// Mitsubishi GX Works2 project: 14.05.24-cascade-2   PLC: FX3G
// Каскад начинается с 2х.

TYPE PUMP : STRUCT
  TurnOn : INT;
  EnableManual : INT;
  OutTask : INT;  (* AO value 0-4000 *)
  Blocked : INT;
  Enable : INT;
  ManualTask : INT;  (* Percent 0.0-100.0 *)
  EnableAuto : INT;
END_STRUCT END_TYPE

// global labels: GVL
VAR_GLOBAL
  giMaxTempr AT R0 : INT;
  gxManual AT M2000 : BOOL;
  gxAuto AT M400 : BOOL;
  gxReset AT M2002 : BOOL;
  gxPump1Enable AT M500 : BOOL;
  gxPump2Enable AT M501 : BOOL;
  gxPump3Enable AT M502 : BOOL;
  gxPump4Enable AT M503 : BOOL;
  gxPump5Enable AT M504 : BOOL;
  gxPump6Enable AT M505 : BOOL;
  arModbus : ARRAY [0..29] OF MB_REG;
  giPSV AT R1 : INT;  (* Set value for pressure 0.00 *)
  giPIDtask AT R2 : INT;
  gxPIDAT AT M2020 : BOOL;
  gxPIDATMode AT M2021 : BOOL;
  gxPump1Manual AT M2009 : BOOL;
  gxPump2Manual AT M2010 : BOOL;
  gxPump3Manual AT M2011 : BOOL;
  gxPump4Manual AT M2012 : BOOL;
  gxPump5Manual AT M2013 : BOOL;
  arPumps : ARRAY [0..4] OF PUMP;
END_VAR
VAR_GLOBAL CONSTANT
  c_PUMPS : INT := 5;
END_VAR
VAR_GLOBAL
  giMaxDiffPressure AT R3 : INT;
  gxPump6Manual AT M2014 : BOOL;
  giMinFlow AT R4 : INT;  (* Если проток больше чем это то включаем полив *)
  giMinPressure AT R5 : INT;  (* Если давление меньше чем это то включаем полив *)
  giMaxPressureRelease AT R6 : INT;
  gxValveManual AT M2015 : BOOL;
  gxErrorJokey AT M2016 : BOOL;
  gxIsAlarm AT M2017 : BOOL;
  gxRecord AT M2018 : BOOL;
  gxResetCounters AT M2019 : BOOL;
END_VAR

// global labels: IO
VAR_GLOBAL
  AI_T_Pump1 AT D0 : INT;
  AI_T_Pump2 AT D1 : INT;
  AI_T_Pump3 AT D2 : INT;
  AI_T_Pump4 AT D3 : INT;
  AI_T_Pump5 AT D4 : INT;
  AI_T_Pump6 AT D5 : INT;
  AI_P_Collector AT D6 : INT;
  AI_P_Filter AT D7 : INT;
  AI_F_Flow AT D8 : INT;
  DI_HighPressure AT X000 : BOOL;
  DI_AU AT X001 : BOOL;
  DI_RKF AT X002 : BOOL;
  DI_T_Panel1_High AT X003 : BOOL;
  DI_T_Panel2_High AT X004 : BOOL;
  DI_FlowPLS AT X005 : BOOL;
  DI_FlowPump1 AT X012 : BOOL;
  DI_FlowPump2 AT X013 : BOOL;
  DI_FlowPump3 AT X014 : BOOL;
  DI_FlowPump4 AT X015 : BOOL;
  DI_FlowPump5 AT X016 : BOOL;
  DI_FlowPump6 AT X017 : BOOL;
  DO_Pump1 AT Y004 : BOOL;
  DO_ResetVFD1 AT Y005 : BOOL;
  DO_Pump2 AT Y006 : BOOL;
  DO_ResetVFD2 AT Y007 : BOOL;
  DO_Pump3 AT Y010 : BOOL;
  DO_ResetVFD3 AT Y011 : BOOL;
  DO_Pump4 AT Y012 : BOOL;
  DO_ResetVFD4 AT Y013 : BOOL;
  DO_Pump5 AT Y014 : BOOL;
  DO_ResetVFD5 AT Y015 : BOOL;
  DO_PumpJok AT Y016 : BOOL;
  DO_ResetVFDJok AT Y017 : BOOL;
  DO_ReleaseValve AT Y020 : BOOL;
  AO_Pump1 AT D8050 : INT;
  AO_Pump2 AT D8051 : INT;
  AO_Pump3 AT D8052 : INT;
  AO_Pump4 AT D8053 : INT;
  AO_Pump5 AT D8054 : INT;
END_VAR

// task INIT (event M8002, interval 0, priority 24): Init
// task PRC (event FALSE, interval T#50ms, priority 29): Process
// task Task_01 (event TRUE, interval 0, priority 31): POU_01
// user libraries (not included): AlarmManger128, Modbus, PumpControl, TimeControl, Utils

PROGRAM Init
VAR
  fbAmInit : AM_INIT;
END_VAR
(* Init PID *) (* Настройка параметров ПИД регулирования *)
R500 := 100; (* Time 1c *)
R501 := 2#0000_0000_0000_0001; (* Heating mode *)
R522 := 1000; (* Output max 100% *)
R523 := 0; (* Output min *)
R525 := 10; (* Delta for Autotune 0.5 bar *)
R526 := R522; (* Autotune output upper value *)
R527 := 0; (* Autotune output lower value *)

(* Start alarm manager data at D3000 *)
AM_D_START := 3000;

(* Temperature sensor 1-6 wire out *)
fbAmInit(iNum := 0, iSeverity := AM_ERROR, iProcess := 1);
fbAmInit(iNum := 1);
fbAmInit(iNum := 2);
fbAmInit(iNum := 3);
fbAmInit(iNum := 4);
fbAmInit(iNum := 5);
(* Pressure sensor wire out *)
fbAmInit(iNum := 6, xLock := 1);
(* Pressure sensor after filter wire out *)
fbAmInit(iNum := 7);
(* Flow meter wire out *)
fbAmInit(iNum := 8);
(* Alarm water level level *)
fbAmInit(iNum := 9);
(* Pump temperature too high *)
fbAmInit(iNum := 10, xLatch := 1, xLock := 0);
fbAmInit(iNum := 11);
fbAmInit(iNum := 12);
fbAmInit(iNum := 13);
fbAmInit(iNum := 14);
fbAmInit(iNum := 15);
(* Pump flow *)
fbAmInit(iNum := 16);
fbAmInit(iNum := 17);
fbAmInit(iNum := 18);
fbAmInit(iNum := 19);
fbAmInit(iNum := 20);
fbAmInit(iNum := 21);

(* Max pressure diff *)
fbAmInit(iNum := 22, xLatch := 1, xLock := 1);
(* High pressure *)
fbAmInit(iNum := 23, xLatch := 0, xLock := 1);
(* High tempr 1 *)
fbAmInit(iNum := 24, xLatch := 1, xLock := 1);
(* High tempr 2 *)
fbAmInit(iNum := 25, xLatch := 1, xLock := 1);
(* RKF *)
fbAmInit(iNum := 26, xLatch := 0, xLock := 1);
(* MB Timeout *)
fbAmInit(iNum := 27, xLatch := 0, xLock := 0);
(* Parametrs all set *)
fbAmInit(iNum := 28, xLatch := 0, xLock := 1);

(* Pump VFD Alarm *)
fbAmInit(iNum := 29, xLatch := 0, xLock := 0);
fbAmInit(iNum := 30);
fbAmInit(iNum := 31);
fbAmInit(iNum := 32);
fbAmInit(iNum := 33);
fbAmInit(iNum := 34);

(* Библиотека драйверов Modbus RTU , ПЛК Coolmay FX3G для управления преобразователями частоты , далее ПЧ *)
arModbus[0].iDev := H1; (* Device address *)
arModbus[0].iRDevNum := 3000; (* R memmory to locate result *)
arModbus[0].iNum := 14; (* Number of registers *)
arModbus[0].iReg := H3000; (* Modbus register *)
arModbus[0].iRF := H3; (* Read function *)
arModbus[0].iWR := MB_READ; (* Read and\or write access *)
arModbus[0].tCycle := T#1000ms; (* How oftent *)

arModbus[1].iDev := H2; (* Device address *)
arModbus[1].iRDevNum := 3020; (* R memmory to locate result *)
arModbus[1].iNum := 14; (* Number of registers *)
arModbus[1].iReg := H3000; (* Modbus register *)
arModbus[1].iRF := H3; (* Read function *)
arModbus[1].iWR := MB_READ; (* Read and\or write access *)
arModbus[1].tCycle := T#1000ms; (* How oftent *)

arModbus[2].iDev := H3; (* Device address *)
arModbus[2].iRDevNum := 3040; (* R memmory to locate result *)
arModbus[2].iNum := 14; (* Number of registers *)
arModbus[2].iReg := H3000; (* Modbus register *)
arModbus[2].iRF := H3; (* Read function *)
arModbus[2].iWR := MB_READ; (* Read and\or write access *)
arModbus[2].tCycle := T#1000ms; (* How oftent *)

arModbus[3].iDev := H4; (* Device address *)
arModbus[3].iRDevNum := 3060; (* R memmory to locate result *)
arModbus[3].iNum := 14; (* Number of registers *)
arModbus[3].iReg := H3000; (* Modbus register *)
arModbus[3].iRF := H3; (* Read function *)
arModbus[3].iWR := MB_READ; (* Read and\or write access *)
arModbus[3].tCycle := T#1000ms; (* How oftent *)

arModbus[4].iDev := H5; (* Device address *)
arModbus[4].iRDevNum := 3080; (* R memmory to locate result *)
arModbus[4].iNum := 14; (* Number of registers *)
arModbus[4].iReg := H3000; (* Modbus register *)
arModbus[4].iRF := H3; (* Read function *)
arModbus[4].iWR := MB_READ; (* Read and\or write access *)
arModbus[4].tCycle := T#1000ms; (* How oftent *)

arModbus[5].iDev := H6; (* Device address *)
arModbus[5].iRDevNum := 3100; (* R memmory to locate result *)
arModbus[5].iNum := 1; (* Number of registers *)
arModbus[5].iReg := H3002; (* Modbus register *)
arModbus[5].iRF := H4; (* Read function *)
arModbus[5].iWR := MB_READ; (* Read and\or write access *)
arModbus[5].tCycle := T#1000ms; (* How oftent *)
END_PROGRAM

PROGRAM POU_01
VAR
  iCount : INT;
  iCountEnabled : INT;
  iCountEbabledAuto : INT;
  iStep : INT;
  xAddOne : BOOL;
  xSubOne : BOOL;
  fbAmBlock : AM_IS_BLOCK;
  xError : BOOL;
  fbAmOrIsOn : AM_ORISON;
  fbReleaseTOF : TOF;
  fbRelease2TOF : TOF;
  iShifter : INT;
  iShifted : INT;
  xAfterAdd : BOOL;
  xFromJokey : BOOL;
  xAfterSub : BOOL;
END_VAR
IF MEP(gxAuto) AND gxPIDAT THEN
	R501 := 2#0000_0000_0011_0001; (* Autotune Step Response *)
	IF NOT gxPIDATMode THEN
		R501 := 2#0000_0000_0111_0001; (* Autotune limit cycle *)
	END_IF;
	gxPIDAT := FALSE;
END_IF;

RST(MEP(gxManual), gxAuto);
RST(MEP(gxAuto), gxManual);

fbAmBlock(iProcessNum := 1, iSeverity := AM_ERROR);
gxIsAlarm := fbAmBlock.Q;

(* IF there is blocking alarm AND we are in auto OR manual OR jokey mode, EXIT it *)
IF fbAmBlock.Q AND iStep <> 10 THEN	iStep := 0; END_IF;

PID(iStep = 30 AND (AI_P_Collector < (giPSV + 50)), giPSV, AI_P_Collector, R500, giPIDTask);

IF MEP(iStep = 30) THEN iShifter := INC5(iShifter); END_IF;
OUT_T(iStep = 30 AND xAfterAdd, TC14, 100);
RST(MEP(TS14), xAfterAdd);

OUT_T(iStep = 30 AND xAfterSub, TC16, 100);
RST(MEP(TS16), xAfterSub);

(*OUT_T(iStep = 30 AND NOT TS15 AND NOT xAfterAdd, TC15, 100);*)

OUT_T(iStep = 35, TC13, 60); (* time to add new pump *)
OUT_T(iStep = 30 AND AI_F_Flow < 200 AND (AI_P_Collector > giMinPressure), TC21, 50); (* to jokey *)

CASE iStep OF
	0: (* Init *)
		gxManual := FALSE;
		FOR iCount := 0 TO 4 DO
			arPumps[iCount].OutTask := 0;
			arPumps[iCount].TurnOn := 0;
			arPumps[iCount].ManualTask := 0;
			arPumps[iCount].EnableAuto := 0;
			arPumps[iCount].EnableManual := 0;
		END_FOR;
		iStep := 10;

	10: (* Idle *) (* *)
		IF gxManual AND NOT fbAmBlock.Q THEN
			iStep := 20;
		END_IF;
		IF gxAuto AND NOT fbAmBlock.Q THEN
			iStep := 30;
		END_IF;

	20: (* Manual *)
        FOR iCount := 0 TO 4 DO
			IF arPumps[iCount].Enable = 0 THEN arPumps[iCount].EnableManual := 0; END_IF;

			arPumps[iCount].TurnOn := BOOL_TO_INT(
				NOT INT_TO_BOOL(arPumps[iCount].Blocked)
				AND INT_TO_BOOL(arPumps[iCount].Enable)
				AND INT_TO_BOOL(arPumps[iCount].EnableManual)
			);

			arPumps[iCount].OutTask := 0;
			IF arPumps[iCount].TurnOn = 1 THEN
				arPumps[iCount].OutTask := SCALE(arPumps[iCount].ManualTask, 0, 1000, 0, 4000);
			END_IF;
		END_FOR;

		IF NOT gxManual THEN iStep := 0; END_IF;

	30: (* Auto CASCADE *)
		(* Once every 10 seconds *)
		iCountEnabled := 0;	 iCountEbabledAuto := 0;
		FOR iCount := 0 TO 4 DO
			IF arPumps[iCount].Enable = 0 THEN arPumps[iCount].EnableAuto := 0; END_IF;
			(* Globally ready pumps for work *)
			IF arPumps[iCount].Enable > 0 AND (arPumps[iCount].Blocked = 0) THEN
				iCountEnabled := iCountEnabled + 1;
			END_IF;

			(* Count currently enabled pumps in cascade *)
			iCountEbabledAuto := iCountEbabledAuto + arPumps[iCount].EnableAuto;
		END_FOR;
		
		(* Add new pump to cascade if PID task > 90.0% and there is a pump available *)
		xAddOne := xFromJokey OR ((giPIDTask > 950) AND (
			(iCountEbabledAuto > 0 AND AI_P_Collector < (giPSV - 100)) OR iCountEbabledAuto = 0
		) AND (iCountEnabled > iCountEbabledAuto));
		(* Subtract pump if task is less than 40.0% or 25 HGz if there are more than 2 pumps enabled *)
		xSubOne := giPIDTask < 780 AND iCountEbabledAuto > 2;
		xFromJokey := FALSE;
		
		IF xAddOne AND NOT xAfterAdd THEN 
			iStep := 35; 
		END_IF;
		
		FOR iCount := 0 TO 4 DO
			iShifted := SHFT(iShifter, iCount);
			IF xSubOne 
				AND NOT xAfterSub 
				AND arPumps[iShifted].Enable > 0 
				AND arPumps[iShifted].Blocked = 0 
				AND arPumps[iShifted].EnableAuto > 0 
			THEN
				arPumps[iShifted].EnableAuto := 0;
				xSubOne := FALSE;
				xAfterSub := TRUE;
			END_IF; 
			
			arPumps[iShifted].TurnOn := BOOL_TO_INT(
				NOT INT_TO_BOOL(arPumps[iShifted].Blocked) 
				AND INT_TO_BOOL(arPumps[iShifted].Enable) 
				AND INT_TO_BOOL(arPumps[iShifted].EnableAuto)
				AND AI_P_Collector < (giPSV + 50)
			);

			arPumps[iShifted].OutTask := 0;
			IF arPumps[iShifted].TurnOn > 0 THEN
				arPumps[iShifted].OutTask := SCALE(giPIDTask, 0, 1000, 0, 4000);
			END_IF;
		END_FOR;
		
		(* TODO condition to switch to Jokey *)
		
		(* IF AI_F_Flow <= giMinFlow THEN *) 
		IF  TS21 THEN 
			FOR iCount := 0 TO 4 DO
				arPumps[iCount].OutTask := 0;
				arPumps[iCount].TurnOn := 0;
				arPumps[iCount].ManualTask := 0;
				arPumps[iCount].EnableAuto := 0;
				arPumps[iCount].EnableManual := 0;
			END_FOR;
			iStep := 40;
		END_IF;

		IF NOT gxAuto OR gxReset THEN iStep := 0; END_IF;
	
	35:
	    iCountEbabledAuto := 0;
	    FOR iCount := 0 TO 4 DO
				iCountEbabledAuto := iCountEbabledAuto + arPumps[iCount].EnableAuto;
	    END_FOR;
	    
		FOR iCount := 0 TO 4 DO
			iShifted := SHFT(iShifter, iCount);
			IF xAddOne AND arPumps[iShifted].Enable > 0 AND arPumps[iShifted].Blocked = 0 AND arPumps[iShifted].EnableAuto = 0 THEN
				arPumps[iShifted].EnableAuto := 1;
				IF iCountEbabledAuto < 1 THEN
					iCountEbabledAuto := iCountEbabledAuto + arPumps[iShifted].EnableAuto;
				ELSE
					xAddOne := FALSE;
				END_IF;
			END_IF; 
			
			arPumps[iShifted].TurnOn := BOOL_TO_INT(
				NOT INT_TO_BOOL(arPumps[iShifted].Blocked) 
				AND INT_TO_BOOL(arPumps[iShifted].Enable) 
				AND INT_TO_BOOL(arPumps[iShifted].EnableAuto)
			);

			arPumps[iShifted].OutTask := 0;
			IF arPumps[iShifted].TurnOn > 0 THEN
				arPumps[iShifted].OutTask := SCALE(750, 0, 1000, 0, 4000);
			END_IF;
		END_FOR;
		
		IF TS13 THEN
			iStep := 30;
			xAfterAdd := TRUE;
		END_IF;

	40: (* jokey in auto *)
        (* AI_F_Flow > giMinFlow AND *)
		IF (AI_P_Collector < giMinPressure) THEN
			iStep := 30;
			xFromJokey := TRUE;
			xAfterAdd := FALSE;
		END_IF;

		IF NOT gxAuto OR gxReset THEN iStep := 0; END_IF;
END_CASE;

gxErrorJokey := FALSE;
fbAmOrIsOn(iNum := 5, Q := gxErrorJokey);
fbAmOrIsOn(iNum := 15, Q := gxErrorJokey);
fbAmOrIsOn(iNum := 21, Q := gxErrorJokey);
fbAmOrIsOn(iNum := 34, Q := gxErrorJokey);
(* Enable Joker if in manual and turned on or auto mode *)
DO_PumpJok := NOT gxErrorJokey AND gxPump6Enable AND (
	(iStep = 20 AND gxPump6Manual) OR (iStep = 40)
);

fbReleaseTOF(IN := (AI_P_Collector > giMaxPressureRelease), PT := T#5s);
fbRelease2TOF(IN := DI_HighPressure, PT := T#15s);
DO_ReleaseValve := fbReleaseTOF.Q OR fbRelease2TOF.Q OR gxValveManual;

AO_Pump1 := arPumps[0].OutTask;
AO_Pump2 := arPumps[1].OutTask;
AO_Pump3 := arPumps[2].OutTask;
AO_Pump4 := arPumps[3].OutTask;
AO_Pump5 := arPumps[4].OutTask;

DO_Pump1 := (arPumps[0].TurnOn > 0);
DO_Pump2 := (arPumps[1].TurnOn > 0);
DO_Pump3 := (arPumps[2].TurnOn > 0);
DO_Pump4 := (arPumps[3].TurnOn > 0);
DO_Pump5 := (arPumps[4].TurnOn > 0);

gxRecord := (DO_Pump1 OR DO_Pump2 OR DO_Pump3 OR DO_Pump4 OR DO_Pump5 OR DO_PumpJok OR TRUE);
END_PROGRAM

PROGRAM Process
VAR
  fbAMSET : AM_SET;
  fbAmReset : AM_RST;
  PortSettings : DWORD;
  fbAmOrIsOn : AM_ORISON;
  xError : BOOL;
END_VAR
IF D8030 = 4984 THEN AI_T_Pump1 := 0; ELSE AI_T_Pump1 := D8030; END_IF;
IF D8031 = 4984 THEN AI_T_Pump2 := 0; ELSE AI_T_Pump2 := D8031; END_IF;
IF D8032 = 4984 THEN AI_T_Pump3 := 0; ELSE AI_T_Pump3 := D8032; END_IF;
IF D8033 = 4984 THEN AI_T_Pump4 := 0; ELSE AI_T_Pump4 := D8033; END_IF;
IF D8034 = 4984 THEN AI_T_Pump5 := 0; ELSE AI_T_Pump5 := D8034; END_IF;
IF D8035 = 4984 THEN AI_T_Pump6 := 0; ELSE AI_T_Pump6 := D8035; END_IF;
IF D8036 = 32760 THEN AI_P_Collector := 0; ELSE AI_P_Collector := SCALE(D8036, 0, 4000, 0, 1600); END_IF;
IF D8037 = 32760 THEN AI_P_Filter := 0; ELSE AI_P_Filter := SCALE(D8037, 0, 4000, 0, 1600); END_IF;
IF D8038 = 32760 THEN AI_F_Flow := 0; ELSE AI_F_Flow := SCALE(D8038, 0, 4000, 0, 8800); END_IF;

(* Analog alarms *) (* Функциональный блок Менеджера Оповещений , далее МО, нулевого уровня значения аналогового сигнала *)
fbAMSET(iNum := 0, xState := (D8030 = 4984));
fbAMSET(iNum := 1, xState := (D8031 = 4984));
fbAMSET(iNum := 2, xState := (D8032 = 4984));
fbAMSET(iNum := 3, xState := (D8033 = 4984));
fbAMSET(iNum := 4, xState := (D8034 = 4984));
fbAMSET(iNum := 5, xState := (D8035 = 4984));
fbAMSET(iNum := 6, xState := (D8036 = 32760));
fbAMSET(iNum := 7, xState := (D8037 = 32760));
fbAMSET(iNum := 8, xState := (D8038 = 32760));
(* Water level too low *)
fbAMSET(iNum := 9, xState := (NOT DI_AU));
(* Pump temperature too high *)
OUT_T((AI_T_Pump1 >= giMaxTempr), TC6, 300);
OUT_T((AI_T_Pump2 >= giMaxTempr), TC7, 300);
OUT_T((AI_T_Pump3 >= giMaxTempr), TC8, 300);
OUT_T((AI_T_Pump4 >= giMaxTempr), TC9, 300);
OUT_T((AI_T_Pump5 >= giMaxTempr), TC10, 300);
OUT_T((AI_T_Pump6 >= giMaxTempr), TC11, 300);
fbAMSET(iNum := 10, xState := TS6);
fbAMSET(iNum := 11, xState := TS7);
fbAMSET(iNum := 12, xState := TS8);
fbAMSET(iNum := 13, xState := TS9);
fbAMSET(iNum := 14, xState := TS10);
fbAMSET(iNum := 15, xState := TS11);
(* Pump flow *)
OUT_T((NOT DI_FlowPump1 AND DO_Pump1), TC0, 600);
OUT_T((NOT DI_FlowPump2 AND DO_Pump2), TC1, 600);
OUT_T((NOT DI_FlowPump3 AND DO_Pump3), TC2, 600);
OUT_T((NOT DI_FlowPump4 AND DO_Pump4), TC3, 600);
OUT_T((NOT DI_FlowPump5 AND DO_Pump5), TC4, 600);
OUT_T((NOT DI_FlowPump6 AND DO_PumpJok), TC5, 6000);
fbAMSET(iNum := 16, xState := TS0);
fbAMSET(iNum := 17, xState := TS1);
fbAMSET(iNum := 18, xState := TS2);
fbAMSET(iNum := 19, xState := TS3);
fbAMSET(iNum := 20, xState := TS4);
fbAMSET(iNum := 21, xState := TS5);

(* Max diff pressure *)
fbAMSET(iNum := 22, xState := (AI_P_Collector - AI_P_Filter) > giMaxDiffPressure);
(* High pressure *)
fbAMSET(iNum := 23, xState := DI_HighPressure);
(* High tempr 1 *)
fbAMSET(iNum := 24, xState := DI_T_Panel1_High);
(* High tempr 2 *)
fbAMSET(iNum := 25, xState := DI_T_Panel2_High);
(* RKF *)
fbAMSET(iNum := 26, xState := NOT DI_RKF);
(* MB Timeout *)
fbAMSET(iNum := 27, xState := FALSE);
(* All parameters set *)
fbAMSET(iNum := 28, xState := (
		giMaxTempr = 0 OR giPSV = 0 OR giMaxDiffPressure = 0 OR
		giMinFlow = 0 OR giMinPressure = 0 OR giMaxPressureRelease = 0 OR
		(NOT gxPump1Enable AND NOT gxPump2Enable AND NOT gxPump3Enable AND NOT gxPump4Enable AND NOT gxPump5Enable)
	)
);

(* Pump VFD alarm from Modbus *)
fbAMSET(iNum := 29, xState := FALSE);
fbAMSET(iNum := 30, xState := FALSE);
fbAMSET(iNum := 31, xState := FALSE);
fbAMSET(iNum := 32, xState := FALSE);
fbAMSET(iNum := 33, xState := FALSE);
fbAMSET(iNum := 34, xState := FALSE);

(* либо датчика минимального потока , либо датчика минимального
давления, либо датчика максимального выходного давления *)
fbAmReset(IN := gxReset);

xError := FALSE;
fbAmOrIsOn(iNum := 29, Q := xError);
DO_ResetVFD1 := gxReset AND xError;

xError := FALSE;
fbAmOrIsOn(iNum := 30, Q := xError);
DO_ResetVFD2 := gxReset;

xError := FALSE;
fbAmOrIsOn(iNum := 31, Q := xError);
DO_ResetVFD3 := gxReset;

xError := FALSE;
fbAmOrIsOn(iNum := 32, Q := xError);
DO_ResetVFD4 := gxReset;

xError := FALSE;
fbAmOrIsOn(iNum := 33, Q := xError);
DO_ResetVFD5 := gxReset;

xError := FALSE;
fbAmOrIsOn(iNum := 34, Q := xError);
DO_ResetVFDJok := gxReset;


IF M8002 OR gxReset THEN (* Если происходит сброс ошибки ПЧ *)
	PortSettings := MB_PORT_SETTINGS(MB_PARITY_EVEN, MB_STOPBIT_1, MB_BPS_19200);
END_IF;
M0 := MB_MASTER_INIT_PORT2(gxReset OR M8002, PortSettings);
(* fbMbProcess(mb_arRegs := arModbus, mb_xEnable := NOT gxReset AND gxReset = FALSE); *)
(* не может принимать значения : gxReset и FALSE *)

HOUR(DO_Pump1, K30000, R5500, M5500);
HOUR(DO_Pump2, K30000, R5502, M5501);
HOUR(DO_Pump3, K30000, R5504, M5502);
HOUR(DO_Pump4, K30000, R5506, M5503);
HOUR(DO_Pump5, K30000, R5508, M5504);
HOUR(DO_PumpJok, K30000, R5510, M5505);
RST(gxResetCounters, R5500);
RST(gxResetCounters, R5502);
RST(gxResetCounters, R5504);
RST(gxResetCounters, R5506);
RST(gxResetCounters, R5508);
RST(gxResetCounters, R5510);
RST(gxResetCounters, gxResetCounters);

xError := FALSE;
fbAmOrIsOn(iNum := 0, Q := xError);
fbAmOrIsOn(iNum := 10, Q := xError);
fbAmOrIsOn(iNum := 16, Q := xError);
fbAmOrIsOn(iNum := 29, Q := xError);
arPumps[0].Blocked := BOOL_TO_INT(xError);
arPumps[0].Enable := BOOL_TO_INT(gxPump1Enable);
arPumps[0].EnableManual := BOOL_TO_INT(gxPump1Manual);

xError := FALSE;
fbAmOrIsOn(iNum := 1, Q := xError);
fbAmOrIsOn(iNum := 11, Q := xError);
fbAmOrIsOn(iNum := 17, Q := xError);
fbAmOrIsOn(iNum := 30, Q := xError);
arPumps[1].Blocked := BOOL_TO_INT(xError);
arPumps[1].Enable := BOOL_TO_INT(gxPump2Enable);
arPumps[1].EnableManual := BOOL_TO_INT(gxPump2Manual);


xError := FALSE;
fbAmOrIsOn(iNum := 2, Q := xError);
fbAmOrIsOn(iNum := 12, Q := xError);
fbAmOrIsOn(iNum := 18, Q := xError);
fbAmOrIsOn(iNum := 31, Q := xError);
arPumps[2].Blocked := BOOL_TO_INT(xError);
arPumps[2].Enable := BOOL_TO_INT(gxPump3Enable);
arPumps[2].EnableManual := BOOL_TO_INT(gxPump3Manual);

xError := FALSE;
fbAmOrIsOn(iNum := 3, Q := xError);
fbAmOrIsOn(iNum := 13, Q := xError);
fbAmOrIsOn(iNum := 19, Q := xError);
fbAmOrIsOn(iNum := 32, Q := xError);
arPumps[3].Blocked := BOOL_TO_INT(xError);
arPumps[3].Enable := BOOL_TO_INT(gxPump4Enable);
arPumps[3].EnableManual := BOOL_TO_INT(gxPump4Manual);

xError := FALSE;
fbAmOrIsOn(iNum := 4, Q := xError);
fbAmOrIsOn(iNum := 14, Q := xError);
fbAmOrIsOn(iNum := 20, Q := xError);
fbAmOrIsOn(iNum := 33, Q := xError);
arPumps[4].Blocked := BOOL_TO_INT(xError);
arPumps[4].Enable := BOOL_TO_INT(gxPump5Enable);
arPumps[4].EnableManual := BOOL_TO_INT(gxPump5Manual);

RST(gxPump1Manual AND NOT gxManual, gxPump1Manual);
RST(gxPump2Manual AND NOT gxManual, gxPump2Manual);
RST(gxPump3Manual AND NOT gxManual, gxPump3Manual);
RST(gxPump4Manual AND NOT gxManual, gxPump4Manual);
RST(gxPump5Manual AND NOT gxManual, gxPump5Manual);
RST(gxPump6Manual AND NOT gxManual, gxPump6Manual);

R4000 := SCALE(giPIDTask, 0, 1000, 0, 100);
END_PROGRAM

FUNCTION INC5
VAR_INPUT
  CUR : INT;
END_VAR
INC5 := INC5 + 1;
IF INC5 > 5 THEN
	INC5 := INC5 - 5;
END_IF;
END_FUNCTION

FUNCTION SHFT
VAR_INPUT
  SHIFTER : INT;
  IDX : INT;
END_VAR
SHFT := SHIFTER + IDX;
IF SHFT > 4 THEN
	SHFT := SHFT - 5;	
END_IF;
END_FUNCTION
